(* IEC 61131-3 sources: axopen.templates/axopen.template.simple/ax/src/Glob, 3 files *)

(* ---- Globals.st ---- *)
NAMESPACE axosimple

    USING AXOpen.Data;
    USING AXOpen.Core;

    {S7.extern=ReadWrite}
    CLASS PUBLIC GlobalContextObjects EXTENDS AxoObject
        VAR PUBLIC
            {#ix-attr:[AXOpen.Data.PersistentAttribute("")]}
            LastTechnologySettings : STRING ;

            Persits         : AxoDataPersistentExchange;
            PS              : axosimple.ProcessData;
            TS              : axosimple.TechnologyData;
            PD              : axosimple.ProcessData;
        END_VAR

        METHOD PUBLIC Run
            VAR_INPUT
                inParent : IAxoContext;
            END_VAR
            THIS.Initialize(inParent);

            TS.Run(THIS);
            PS.Run(THIS);
            PD.Run(THIS);
            Persits.Run(THIS);

        END_METHOD

    END_CLASS
END_NAMESPACE

(* ---- ProcessData.st ---- *)
NAMESPACE axosimple
    {S7.extern=ReadWrite}
    CLASS ProcessData EXTENDS AXOpen.Data.AxoDataFragmentExchange
        VAR PUBLIC
            {#ix-attr:[AXOpen.Data.AxoDataFragmentAttribute]}
            Entity : SharedDataExchange;

            // Units data - You can use snippet unitAddProcessData

        END_VAR
    END_CLASS
END_NAMESPACE

(* ---- TechnologyData.st ---- *)
NAMESPACE axosimple
    {S7.extern=ReadWrite}
    CLASS TechnologyData EXTENDS AXOpen.Data.AxoDataFragmentExchange
        VAR PUBLIC
            {#ix-attr:[AXOpen.Data.AxoDataFragmentAttribute]}
            Common : TechnologySharedDataExchange;

            // Units data - snippet unitAddTechnologyData

        END_VAR
    END_CLASS
END_NAMESPACE
